// TIA Portal V20 export
DATA_BLOCK "instFB_AutoCtrl_5Pts"   // DB23
VERSION : 1.1
// Instance DB for FB_AutoCtrl_5Pts (Phase 4a, 2026-05-21). Huashili-pattern CASE auto FB; replaces FB_AutoCtrl_ABCDE. DB number may be auto-assigned by TIA on import.
// stored: InstanceOfName FB_AutoCtrl_5Pts, InstanceOfType FB
"FB_AutoCtrl_5Pts"
   // VAR
   //    pts { S7_SetPoint := 'True'} : Array[1..5] of "UDT_typePoint5";
   //    statTargetPos : "UDT_typePoint5";
   //    statPointIdx : Int;
   //    sRTRIGInitPath { S7_SetPoint := 'True'} : R_TRIG;
   //    sRTRIGStart { S7_SetPoint := 'True'} : R_TRIG;
   //    sRTRIGStop { S7_SetPoint := 'True'} : R_TRIG;
   //    sRTRIGAlarm { S7_SetPoint := 'True'} : R_TRIG;
   //    sRTRIGPause { S7_SetPoint := 'True'} : R_TRIG;
   //    statStepBeforePause : Int;
   // END_VAR
BEGIN
END_DATA_BLOCK
